FUNCTION_BLOCK FB_System_FBT_Ablaufsteuerung
VAR_IN_OUT
	Zustand			: ST_System_FBT_Zustand;
	Stellwert			: ST_System_FBT_Stellwert;
	Steuerung			: ST_System_FBT_Steuerung;
END_VAR
VAR_INPUT
	Zustand_Pumpe			: ST_PU_Zustand;
	Zustand_Regelventil		: ST_RV_Zustand;
END_VAR
VAR_OUTPUT
END_VAR
VAR
END_VAR

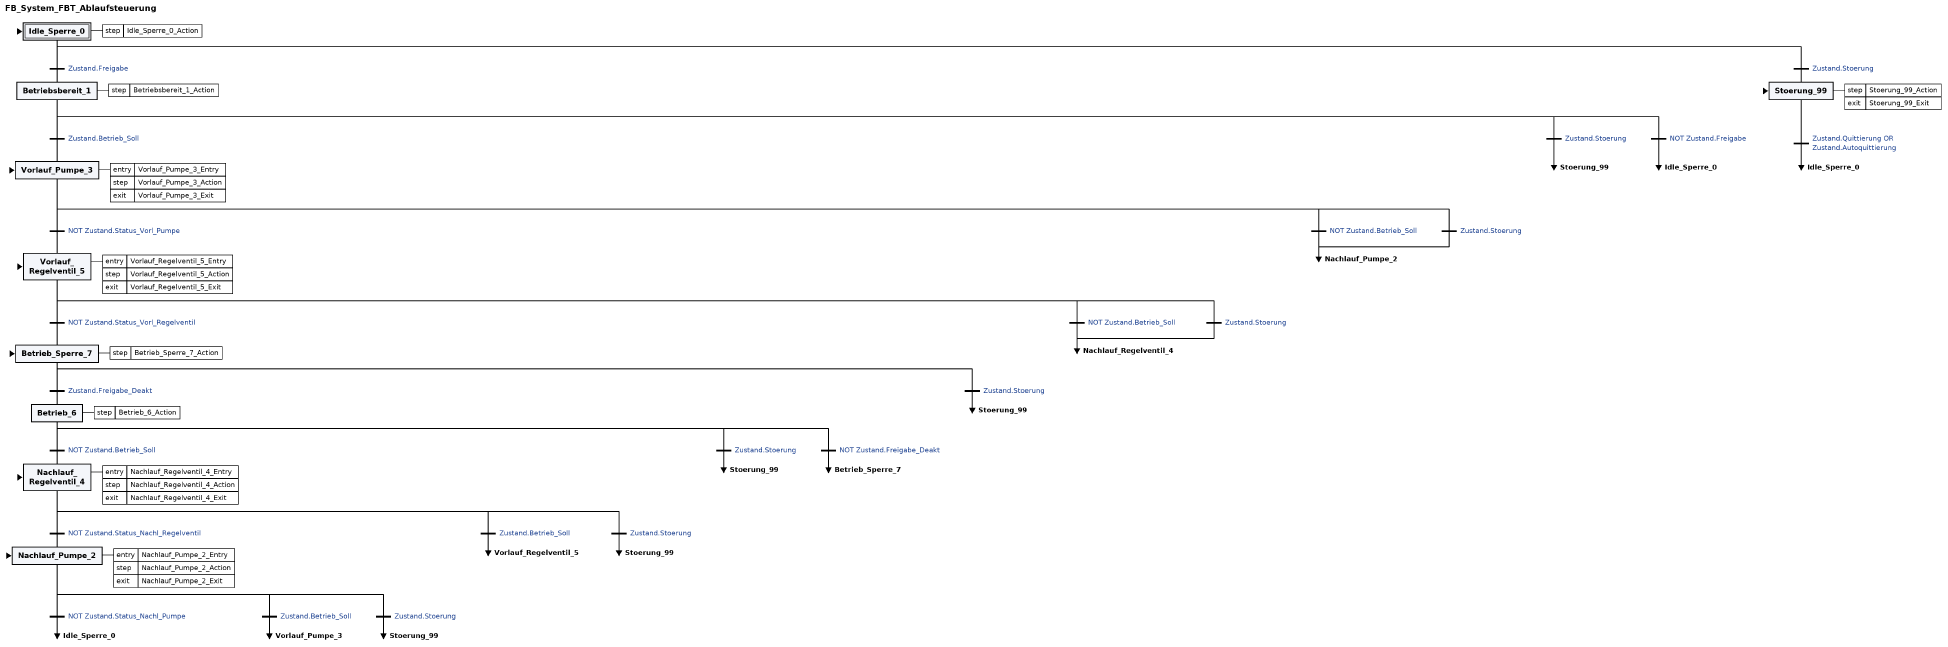
INITIAL_STEP Idle_Sperre_0:
    Idle_Sperre_0_Action(N);  // step action
END_STEP
TRANSITION FROM Idle_Sperre_0 TO Betriebsbereit_1
    := Zustand.Freigabe;
END_TRANSITION
TRANSITION FROM Idle_Sperre_0 TO Stoerung_99
    := Zustand.Stoerung;
END_TRANSITION
STEP Stoerung_99:
    Stoerung_99_Action(N);  // step action
    Stoerung_99_Exit(P0);  // exit action
END_STEP
TRANSITION FROM Stoerung_99 TO Idle_Sperre_0
    := Zustand.Quittierung OR Zustand.Autoquittierung;
END_TRANSITION
STEP Betriebsbereit_1:
    Betriebsbereit_1_Action(N);  // step action
END_STEP
TRANSITION FROM Betriebsbereit_1 TO Vorlauf_Pumpe_3
    := Zustand.Betrieb_Soll;
END_TRANSITION
TRANSITION FROM Betriebsbereit_1 TO Stoerung_99
    := Zustand.Stoerung;
END_TRANSITION
TRANSITION FROM Betriebsbereit_1 TO Idle_Sperre_0
    := NOT Zustand.Freigabe;
END_TRANSITION
STEP Vorlauf_Pumpe_3:
    Vorlauf_Pumpe_3_Entry(P1);  // entry action
    Vorlauf_Pumpe_3_Action(N);  // step action
    Vorlauf_Pumpe_3_Exit(P0);  // exit action
END_STEP
TRANSITION FROM Vorlauf_Pumpe_3 TO Vorlauf_Regelventil_5
    := NOT Zustand.Status_Vorl_Pumpe;
END_TRANSITION
TRANSITION FROM Vorlauf_Pumpe_3 TO Nachlauf_Pumpe_2
    := NOT Zustand.Betrieb_Soll;
END_TRANSITION
TRANSITION FROM Vorlauf_Pumpe_3 TO Nachlauf_Pumpe_2
    := Zustand.Stoerung;
END_TRANSITION
STEP Vorlauf_Regelventil_5:
    Vorlauf_Regelventil_5_Entry(P1);  // entry action
    Vorlauf_Regelventil_5_Action(N);  // step action
    Vorlauf_Regelventil_5_Exit(P0);  // exit action
END_STEP
TRANSITION FROM Vorlauf_Regelventil_5 TO Betrieb_Sperre_7
    := NOT Zustand.Status_Vorl_Regelventil;
END_TRANSITION
TRANSITION FROM Vorlauf_Regelventil_5 TO Nachlauf_Regelventil_4
    := NOT Zustand.Betrieb_Soll;
END_TRANSITION
TRANSITION FROM Vorlauf_Regelventil_5 TO Nachlauf_Regelventil_4
    := Zustand.Stoerung;
END_TRANSITION
STEP Betrieb_Sperre_7:
    Betrieb_Sperre_7_Action(N);  // step action
END_STEP
TRANSITION FROM Betrieb_Sperre_7 TO Betrieb_6
    := Zustand.Freigabe_Deakt;
END_TRANSITION
TRANSITION FROM Betrieb_Sperre_7 TO Stoerung_99
    := Zustand.Stoerung;
END_TRANSITION
STEP Betrieb_6:
    Betrieb_6_Action(N);  // step action
END_STEP
TRANSITION FROM Betrieb_6 TO Nachlauf_Regelventil_4
    := NOT Zustand.Betrieb_Soll;
END_TRANSITION
TRANSITION FROM Betrieb_6 TO Stoerung_99
    := Zustand.Stoerung;
END_TRANSITION
TRANSITION FROM Betrieb_6 TO Betrieb_Sperre_7
    := NOT Zustand.Freigabe_Deakt;
END_TRANSITION
STEP Nachlauf_Regelventil_4:
    Nachlauf_Regelventil_4_Entry(P1);  // entry action
    Nachlauf_Regelventil_4_Action(N);  // step action
    Nachlauf_Regelventil_4_Exit(P0);  // exit action
END_STEP
TRANSITION FROM Nachlauf_Regelventil_4 TO Nachlauf_Pumpe_2
    := NOT Zustand.Status_Nachl_Regelventil;
END_TRANSITION
TRANSITION FROM Nachlauf_Regelventil_4 TO Vorlauf_Regelventil_5
    := Zustand.Betrieb_Soll;
END_TRANSITION
TRANSITION FROM Nachlauf_Regelventil_4 TO Stoerung_99
    := Zustand.Stoerung;
END_TRANSITION
STEP Nachlauf_Pumpe_2:
    Nachlauf_Pumpe_2_Entry(P1);  // entry action
    Nachlauf_Pumpe_2_Action(N);  // step action
    Nachlauf_Pumpe_2_Exit(P0);  // exit action
END_STEP
TRANSITION FROM Nachlauf_Pumpe_2 TO Idle_Sperre_0
    := NOT Zustand.Status_Nachl_Pumpe;
END_TRANSITION
TRANSITION FROM Nachlauf_Pumpe_2 TO Vorlauf_Pumpe_3
    := Zustand.Betrieb_Soll;
END_TRANSITION
TRANSITION FROM Nachlauf_Pumpe_2 TO Stoerung_99
    := Zustand.Stoerung;
END_TRANSITION

ACTION Betrieb_6_Action:
(* Stellwert setzen *)
Stellwert.Anford_Pumpe		:= TRUE;
Stellwert.Anford_Regelventil		:= TRUE;

(* Zustand setzen *)
Zustand.Betrieb				:= TRUE;
Zustand.Status				:= E_System_FBT_Zustand_Status_Betrieb;
END_ACTION

ACTION Betrieb_Sperre_7_Action:
(* Stellwert setzen *)
Stellwert.Anford_Pumpe		:= TRUE;
Stellwert.Anford_Regelventil		:= TRUE;

(* Zustand setzen *)
Zustand.Betrieb				:= TRUE;
Zustand.Status				:= E_System_FBT_Zustand_Status_Betrieb_Sperre;
END_ACTION

ACTION Betriebsbereit_1_Action:
(* Stellwert setzen *)
Stellwert.Anford_Pumpe	:= FALSE;
Stellwert.Anford_Regelventil	:= FALSE;

(* Zustand setzen *)
Zustand.Betrieb			:= FALSE;
Zustand.Status			:= E_System_FBT_Zustand_Status_Betriebsbereit;
END_ACTION

ACTION Idle_Sperre_0_Action:
(* Stellwert setzen *)
Stellwert.Anford_Pumpe	:= FALSE;
Stellwert.Anford_Regelventil	:= FALSE;

(* Zustand setzen *)
Zustand.Betrieb			:= FALSE;
Zustand.Status			:= E_System_FBT_Zustand_Status_Idle_Sperre;

(* Quittierungszustand auf False setzen, damit das System bei einer erneuten Störung nicht direkt wieder angeschaltet wird *)
Steuerung.Quittierung	:= FALSE;
END_ACTION

ACTION Nachlauf_Pumpe_2_Action:
(* Stellwert setzen *)
Stellwert.Anford_Pumpe		:= FALSE;
Stellwert.Anford_Regelventil		:= FALSE;

(* Zustand setzen *)
Zustand.Betrieb				:= FALSE;
Zustand.Status				:= E_System_FBT_Zustand_Status_Nachl_Pumpe;
Zustand.Status_Nachl_Pumpe	:= Zustand_Pumpe.Betrieb OR Zustand_Pumpe.Status_Nachl;
END_ACTION

ACTION Nachlauf_Pumpe_2_Entry:
Zustand.Status_Nachl_Pumpe	:= TRUE;
END_ACTION

ACTION Nachlauf_Pumpe_2_Exit:
Zustand.Status_Nachl_Pumpe	:= FALSE;
END_ACTION

ACTION Nachlauf_Regelventil_4_Action:
(* Stellwert setzen *)
Stellwert.Anford_Pumpe		:= TRUE;
Stellwert.Anford_Regelventil		:= FALSE;

(* Zustand setzen *)
Zustand.Betrieb					:= FALSE;
Zustand.Status					:= E_System_FBT_Zustand_Status_Nachl_Regelventil;
Zustand.Status_Nachl_Regelventil	:= Zustand_Regelventil.Betrieb OR Zustand_Regelventil.Status_Nachl;
END_ACTION

ACTION Nachlauf_Regelventil_4_Entry:
Zustand.Status_Nachl_Regelventil		:= TRUE;
END_ACTION

ACTION Nachlauf_Regelventil_4_Exit:
Zustand.Status_Nachl_Regelventil		:= FALSE;
END_ACTION

ACTION Stoerung_99_Action:
(* Stellwert setzen *)
Stellwert.Anford_Pumpe	:= FALSE;
Stellwert.Anford_Regelventil	:= FALSE;

(* Zustand setzen *)
Zustand.Betrieb			:= FALSE;
Zustand.Stoerung			:= TRUE;
Zustand.Status			:= E_System_FBT_Zustand_Status_Stoerung;
END_ACTION

ACTION Stoerung_99_Exit:
Zustand.Stoerung	:= FALSE;
END_ACTION

ACTION Vorlauf_Pumpe_3_Action:
(* Stellwert setzen *)
Stellwert.Anford_Pumpe		:= TRUE;
Stellwert.Anford_Regelventil		:= FALSE;

(* Zustand setzen *)
Zustand.Betrieb				:= FALSE;
Zustand.Status				:= E_System_FBT_Zustand_Status_Vorl_Pumpe;
Zustand.Status_Vorl_Pumpe	:= NOT(Zustand_Pumpe.Betrieb AND NOT Zustand_Pumpe.Status_Vorl);
END_ACTION

ACTION Vorlauf_Pumpe_3_Entry:
Zustand.Status_Vorl_Pumpe	:= TRUE;
END_ACTION

ACTION Vorlauf_Pumpe_3_Exit:
Zustand.Status_Vorl_Pumpe	:= FALSE;
END_ACTION

ACTION Vorlauf_Regelventil_5_Action:
(* Stellwert setzen *)
Stellwert.Anford_Pumpe		:= TRUE;
Stellwert.Anford_Regelventil		:= TRUE;

(* Zustand setzen *)
Zustand.Betrieb				:= FALSE;
Zustand.Status				:= E_System_FBT_Zustand_Status_Vorl_Regelventil;
Zustand.Status_Vorl_Regelventil	:= NOT(Zustand_Regelventil.Betrieb AND NOT Zustand_Regelventil.Status_Vorl);
END_ACTION

ACTION Vorlauf_Regelventil_5_Entry:
Zustand.Status_Vorl_Regelventil	:= TRUE;
END_ACTION

ACTION Vorlauf_Regelventil_5_Exit:
Zustand.Status_Vorl_Regelventil		:= FALSE;
END_ACTION

END_FUNCTION_BLOCK

(* stored: Version 1.1.0.1, ProductVersion 3.1.4024.9
   POU FB_System_FBT_Ablaufsteuerung: Id {16dd7999-5125-462e-bfc0-8d62314e32b8}, SpecialFunc None
   Action Betrieb_6_Action: Id {3ffc9d38-d786-426d-a13c-161b9cc62cad}
   Action Betrieb_Sperre_7_Action: Id {5a395964-377e-466d-967d-0433809de537}
   Action Betriebsbereit_1_Action: Id {7c2e8059-1c24-40ec-bdb3-45e2e39d214d}
   Action Idle_Sperre_0_Action: Id {c52f5f96-c9fe-496f-99a1-5254034e171a}
   Action Nachlauf_Pumpe_2_Action: Id {a6c23a43-f173-4164-83a6-3476440e473a}
   Action Nachlauf_Pumpe_2_Entry: Id {3bade33c-53e2-470e-aa22-f67691eba5f7}
   Action Nachlauf_Pumpe_2_Exit: Id {6931c2bc-eb9f-430f-afd0-bb7062efe6bf}
   Action Nachlauf_Regelventil_4_Action: Id {5c40f563-4b6c-4394-91ca-f3ce30a179c1}
   Action Nachlauf_Regelventil_4_Entry: Id {f458cc89-a55d-4db5-bb59-5d33aa258319}
   Action Nachlauf_Regelventil_4_Exit: Id {f03192a3-2d5e-4c47-81a9-a5132735cdfd}
   Action Stoerung_99_Action: Id {9ac4aeff-5245-4be4-861f-efb8164d9517}
   Action Stoerung_99_Exit: Id {20e5a1f8-e0a5-4433-bec0-94650e56472d}
   Action Vorlauf_Pumpe_3_Action: Id {3f22a0be-324a-4899-b47c-8f7275934a3c}
   Action Vorlauf_Pumpe_3_Entry: Id {6a910fad-273a-4d46-812b-9a618237e33e}
   Action Vorlauf_Pumpe_3_Exit: Id {c8611bd1-c56a-4867-a026-639457915222}
   Action Vorlauf_Regelventil_5_Action: Id {62942221-5a10-4a22-a3c6-8a8afc1f7962}
   Action Vorlauf_Regelventil_5_Entry: Id {9e34167d-e4e2-484c-b5da-efa1ff172474}
   Action Vorlauf_Regelventil_5_Exit: Id {0f780304-b81a-493c-9827-7d38a5b0e63a} *)
